// TIA Portal V18 export
FUNCTION_BLOCK "HOOTER"   // FB5, FBD
{ S7_Optimized_Access := 'TRUE' }
VERSION : 0.1
// stored: AutoNumber true, IsIECCheckEnabled false, IsRetainMemResEnabled false, MemoryReserve 100, SetENOAutomatically false, UDAEnableTagReadback false
   VAR_INPUT
      COND1 : Bool;
      COND2 : Bool;
      COND3 : Bool;
      COND4 : Bool;
      COND5 : Bool;
      COND6 : Bool;
      COND7 : Bool;
      COND8 : Bool;
      COND9 : Bool;
      COND10 : Bool;
      HOOTER_DI : Bool;
   END_VAR
   VAR_OUTPUT
      HOOTER_HMI : Bool;
      HOOTER_DO : Bool;
   END_VAR
   VAR_IN_OUT
      ACK : Bool;
   END_VAR
   VAR
      RS1 : Bool;
      RS2 : Bool;
      RS3 : Bool;
      RS4 : Bool;
      RS5 : Bool;
      RS6 : Bool;
      RS7 : Bool;
      RS8 : Bool;
      RS9 : Bool;
      RS10 : Bool;
   END_VAR
BEGIN

REGION Network 1
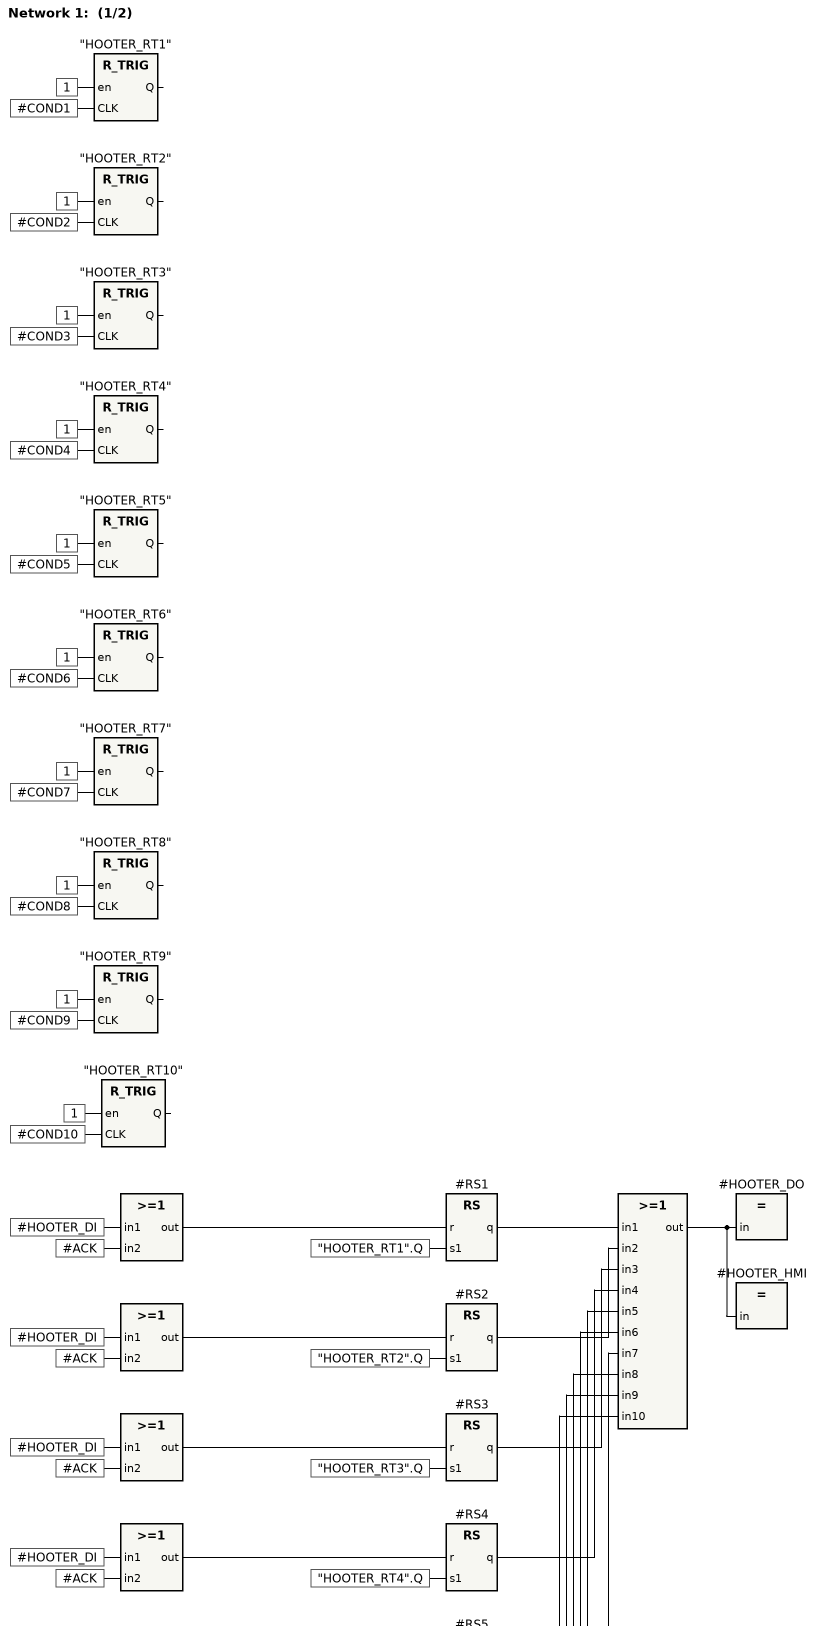
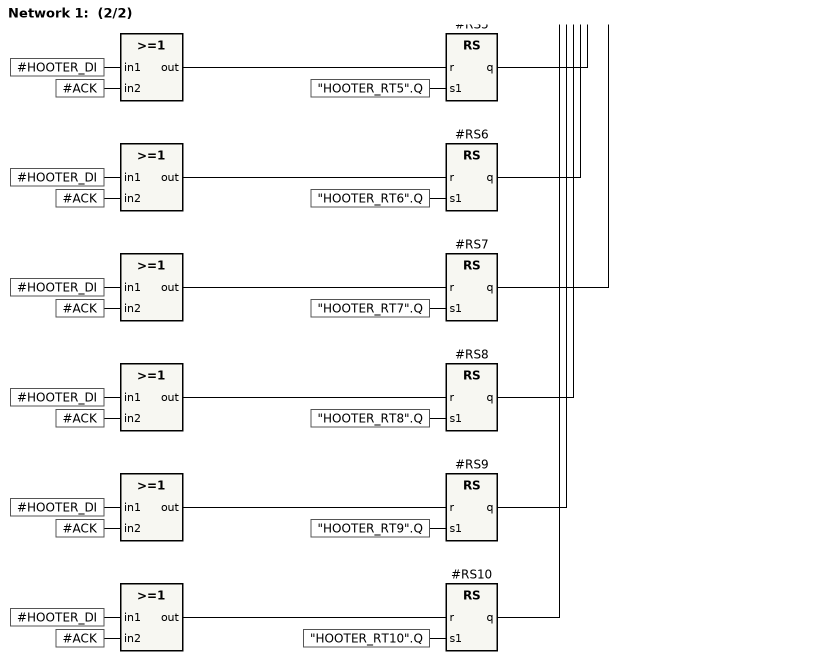
   IF 1 THEN
       "HOOTER_RT1"(CLK := #COND1);   // R_TRIG
       "HOOTER_RT2"(CLK := #COND2);   // R_TRIG
       "HOOTER_RT3"(CLK := #COND3);   // R_TRIG
       "HOOTER_RT4"(CLK := #COND4);   // R_TRIG
       "HOOTER_RT5"(CLK := #COND5);   // R_TRIG
       "HOOTER_RT6"(CLK := #COND6);   // R_TRIG
       "HOOTER_RT7"(CLK := #COND7);   // R_TRIG
       "HOOTER_RT8"(CLK := #COND8);   // R_TRIG
       "HOOTER_RT9"(CLK := #COND9);   // R_TRIG
       "HOOTER_RT10"(CLK := #COND10);   // R_TRIG
   END_IF;
   IF #HOOTER_DI OR #ACK THEN
       #RS1 := FALSE;   // RS flip-flop
   END_IF;
   IF "HOOTER_RT1".Q THEN #RS1 := TRUE; END_IF;
   IF #HOOTER_DI OR #ACK THEN
       #RS2 := FALSE;   // RS flip-flop
   END_IF;
   IF "HOOTER_RT2".Q THEN #RS2 := TRUE; END_IF;
   IF #HOOTER_DI OR #ACK THEN
       #RS3 := FALSE;   // RS flip-flop
   END_IF;
   IF "HOOTER_RT3".Q THEN #RS3 := TRUE; END_IF;
   IF #HOOTER_DI OR #ACK THEN
       #RS4 := FALSE;   // RS flip-flop
   END_IF;
   IF "HOOTER_RT4".Q THEN #RS4 := TRUE; END_IF;
   IF #HOOTER_DI OR #ACK THEN
       #RS5 := FALSE;   // RS flip-flop
   END_IF;
   IF "HOOTER_RT5".Q THEN #RS5 := TRUE; END_IF;
   IF #HOOTER_DI OR #ACK THEN
       #RS6 := FALSE;   // RS flip-flop
   END_IF;
   IF "HOOTER_RT6".Q THEN #RS6 := TRUE; END_IF;
   IF #HOOTER_DI OR #ACK THEN
       #RS7 := FALSE;   // RS flip-flop
   END_IF;
   IF "HOOTER_RT7".Q THEN #RS7 := TRUE; END_IF;
   IF #HOOTER_DI OR #ACK THEN
       #RS8 := FALSE;   // RS flip-flop
   END_IF;
   IF "HOOTER_RT8".Q THEN #RS8 := TRUE; END_IF;
   IF #HOOTER_DI OR #ACK THEN
       #RS9 := FALSE;   // RS flip-flop
   END_IF;
   IF "HOOTER_RT9".Q THEN #RS9 := TRUE; END_IF;
   IF #HOOTER_DI OR #ACK THEN
       #RS10 := FALSE;   // RS flip-flop
   END_IF;
   IF "HOOTER_RT10".Q THEN #RS10 := TRUE; END_IF;
   #HOOTER_DO := #RS1 OR #RS2 OR #RS3 OR #RS4 OR #RS5 OR #RS6 OR #RS7 OR #RS8 OR #RS9 OR #RS10;
   #HOOTER_HMI := #HOOTER_DO;
END_REGION
END_FUNCTION_BLOCK
